// TIA Portal V17 export
// export: Created 2022-07-20T06:59:49.2004828Z, ExportSetting WithDefaults, DisplayName Totally Integrated Automation Portal, DisplayVersion V17, DisplayName TIA Portal Openness, DisplayVersion V17, DisplayName TIA Portal Version Control Interface, DisplayVersion V17, DisplayName SINAMICS Startdrive Advanced, DisplayVersion V17, DisplayName SINAMICS Startdrive G130, G150, S120, S150, SINAMICS MV, S210, DisplayVersion V17, DisplayName SINAMICS Startdrive G110M, G120, G120C, G120D, G120P, G115D, DisplayVersion V17, DisplayName STEP 7 Professional, DisplayVersion V17, DisplayName STEP 7 Safety, DisplayVersion V17, DisplayName WinCC Advanced, DisplayVersion V17
FUNCTION_BLOCK "FB10300_TM_Pulse"   // FB10300, LAD
TITLE = FB10030_TM_Pulse
{ S7_Optimized_Access := 'TRUE' }
AUTHOR : Anirouddh
FAMILY : 1030_SIEMENS
VERSION : 1.0
// Release note : 
// 1.0 - Feature developped
// 
// Todo: 
// - If necessary, complete thre static TM_Pulse structure with the QLMN_HLM & QLMN_LLM to verify that the set value is bounded within the limits
// stored: AutoNumber false, IsIECCheckEnabled false, IsRetainMemResEnabled false, MemoryReserve 100, SetENOAutomatically false, UDAEnableTagReadback false
   VAR_INPUT
      Channel0_SW_Enable : Bool;
      Channel0_Reset_Error : Bool;
      Channel0_Frequency : Real;
      Channel0_Dir : Bool;
      Channel1_SW_Enable : Bool;
      Channel1_Reset_Error : Bool;
      Channel1_Frequency : Real;
      Channel1_Dir : Bool;
      HW_TM_Puls : HW_SUBMODULE;
   END_VAR
   VAR_OUTPUT
      Channel0_Ready : Bool;
      Channel0_SW_Enabled : Bool;
      Channel0_Enable : Bool;
      Channel0_Error : Bool;
      Channel0_DQA : Bool;
      Channel0_Output_Dir : Bool;
      Channel1_Ready : Bool;
      Channel1_SW_Enabled : Bool;
      Channel1_Enable : Bool;
      Channel1_Error : Bool;
      Channel1_DQA : Bool;
      Channel1_Output_Dir : Bool;
   END_VAR
   VAR
      Input_Channel : Array[0..1] of Struct
         ERR_STS1 : Struct
            ERR_PWR : Bool;
            ERR_24V : Bool;
            ERR_LD : Bool;
            ERR_PULSE : Bool;
            ERR_DQA : Bool;
            ERR_DQB : Bool;
            ERR_OUT_VALUE : Bool;
            ERR_SLOT_VAL : Bool;
            Reserved_Bit0 : Bool;
            Reserved_Bit1 : Bool;
            STS_LD_SLOT : Bool;
            Reserved_Bit3 : Bool;
            STS_READY : Bool;
            STS_SW_ENABLE : Bool;
            Reserved_Bit6 : Bool;
            Reserved_Bit7 : Bool;
         END_STRUCT;
         STS2_CNT : Struct
            STS_ENABLE : Bool;
            STS_DQA : Bool;
            STS_DQB : Bool;
            STS_DI : Bool;
            STS_DITHER : Bool;
            Reserved_Bit5 : Bool;
            Reserved_Bit6 : Bool;
            Reserved_Bit7 : Bool;
            SEQ_CNT : Byte;
         END_STRUCT;
         Measured_Current : Word;
         Reserve : Word;
      END_STRUCT;
      Output_Channel : Array[0..1] of Struct
         Output_Value : DWord;
         Slot : DWord;
         Mode_Cmd : Struct
            LD_SLOT_0 : Bool;
            LD_SLOT_1 : Bool;
            LD_SLOT_2 : Bool;
            LD_SLOT_3 : Bool;
            MODE_SLOT : Bool;
            Reserved_Bit5 : Bool;
            Reserved_Bit6 : Bool;
            Reserved_Bit7 : Bool;
            SW_ENABLE : Bool;
            TM_CTRL_DQ : Bool;
            Reserved_Bit2 : Bool;
            SET_DQA : Bool;
            SET_DQB : Bool;
            DITHER : Bool;
            Reserved_Bit8 : Bool;
            Reserved_Bit9 : Bool;
         END_STRUCT;
         Reset : Struct
            RES_ERROR : Bool;
            Reserved_bit1 : Bool;
            Reserved_Bit2 : Bool;
            Reserved_Bit3 : Bool;
            Reserved_Bit4 : Bool;
            Reserved_Bit5 : Bool;
            Reserved_Bit6 : Bool;
            Reserved_Bit7 : Bool;
            Reserved_Bit8 : Bool;
            Reserved_Bit9 : Bool;
            Reserved_Bit10 : Bool;
            Reserved_Bit11 : Bool;
            Reserved_Bit12 : Bool;
            Reserved_Bit13 : Bool;
            Reserved_Bit14 : Bool;
            Reserved_Bit15 : Bool;
         END_STRUCT;
      END_STRUCT;
      RET_VAL_DPRD_DAT : Int;
      RET_VAL_DPWD_DAT : Int;
   END_VAR
BEGIN

REGION Network 1: Read data from TM_Pulse
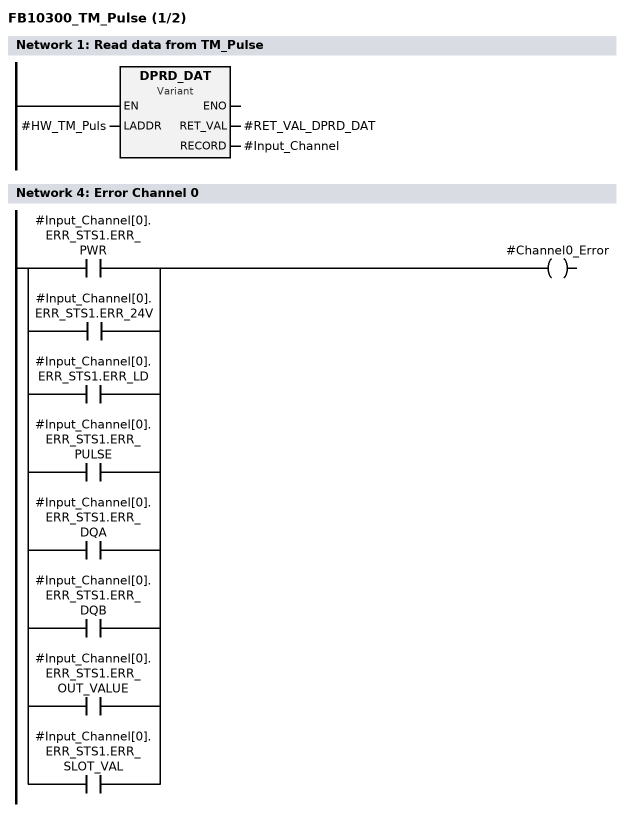
   RUNG wire#powerrail
      { S7_Templates := "[ptr_type := Variant, laddr_type := HW_IO]" } DPRD_DAT(LADDR := #HW_TM_Puls, RET_VAL => #RET_VAL_DPRD_DAT, RECORD => #Input_Channel)
   END_RUNG
   // the same network as SCL:
   #RET_VAL_DPRD_DAT := DPRD_DAT(LADDR := #HW_TM_Puls, RECORD => #Input_Channel);
END_REGION

REGION Network 2 (SCL): Command Channel 0
   #Output_Channel[0].Mode_Cmd.SW_ENABLE := #Channel0_SW_Enable; //Command SW_ENABLE Channel 0
   #Output_Channel[0].Reset.RES_ERROR := #Channel0_Reset_Error; // Command RES_ERROR Channel 0
   #Output_Channel[0].Mode_Cmd.TM_CTRL_DQ := TRUE; //Command TM_CTRL_DQ Channel 0 (The module creates the pulse sequence automatically)
   #Channel0_Output_Dir := #Channel0_Dir; //Command direction Channel 0
   #Output_Channel[0].Output_Value := REAL_TO_DWORD(#Channel0_Frequency); //Command frequence Channel 0

   #Channel0_Ready := #Input_Channel[0].ERR_STS1.STS_READY; //Ready Channel 0
   #Channel0_SW_Enabled := #Input_Channel[0].ERR_STS1.STS_SW_ENABLE; //SW_Enable Channel 0
   #Channel0_Enable := #Input_Channel[0].STS2_CNT.STS_ENABLE; //Enable Channel 0
   #Channel0_DQA := #Input_Channel[0].STS2_CNT.STS_DQA; //DQA Channel 0
END_REGION

REGION Network 3 (SCL): Command Channel 1
   #Output_Channel[1].Mode_Cmd.SW_ENABLE := #Channel1_SW_Enable; //Command SW_ENABLE Channel 1
   #Output_Channel[1].Reset.RES_ERROR := #Channel1_Reset_Error; //Command RES_ERROR Channel 1
   #Output_Channel[1].Mode_Cmd.TM_CTRL_DQ := TRUE; //Command TM_CTRL_DQ Channel 1 (The module creates the pulse sequence automatically)
   #Channel1_Output_Dir := #Channel1_Dir; //Command direction Channel 1
   #Output_Channel[1].Output_Value := REAL_TO_DWORD(#Channel1_Frequency); //Command frequence Channel 1

   #Channel1_Ready := #Input_Channel[1].ERR_STS1.STS_READY; //Ready Channel 1
   #Channel1_SW_Enabled := #Input_Channel[1].ERR_STS1.STS_SW_ENABLE; //SW_Enable Channel 1
   #Channel1_Enable := #Input_Channel[1].STS2_CNT.STS_ENABLE; //Enable Channel 1
   #Channel1_DQA := #Input_Channel[1].STS2_CNT.STS_DQA; //DQA Channel 1
END_REGION

REGION Network 4: Error Channel 0
   RUNG wire#powerrail
      Contact( #Input_Channel[0].ERR_STS1.ERR_PWR )
      wire#w1
      Coil( #Channel0_Error )
   END_RUNG
   RUNG wire#powerrail
      Contact( #Input_Channel[0].ERR_STS1.ERR_24V )
   END_RUNG wire#w1
   RUNG wire#powerrail
      Contact( #Input_Channel[0].ERR_STS1.ERR_LD )
   END_RUNG wire#w1
   RUNG wire#powerrail
      Contact( #Input_Channel[0].ERR_STS1.ERR_PULSE )
   END_RUNG wire#w1
   RUNG wire#powerrail
      Contact( #Input_Channel[0].ERR_STS1.ERR_DQA )
   END_RUNG wire#w1
   RUNG wire#powerrail
      Contact( #Input_Channel[0].ERR_STS1.ERR_DQB )
   END_RUNG wire#w1
   RUNG wire#powerrail
      Contact( #Input_Channel[0].ERR_STS1.ERR_OUT_VALUE )
   END_RUNG wire#w1
   RUNG wire#powerrail
      Contact( #Input_Channel[0].ERR_STS1.ERR_SLOT_VAL )
   END_RUNG wire#w1
   // the same network as SCL:
   #Channel0_Error := #Input_Channel[0].ERR_STS1.ERR_PWR OR #Input_Channel[0].ERR_STS1.ERR_24V OR #Input_Channel[0].ERR_STS1.ERR_LD OR #Input_Channel[0].ERR_STS1.ERR_PULSE OR #Input_Channel[0].ERR_STS1.ERR_DQA OR #Input_Channel[0].ERR_STS1.ERR_DQB OR #Input_Channel[0].ERR_STS1.ERR_OUT_VALUE OR #Input_Channel[0].ERR_STS1.ERR_SLOT_VAL;
END_REGION

REGION Network 5: Error Channel 1
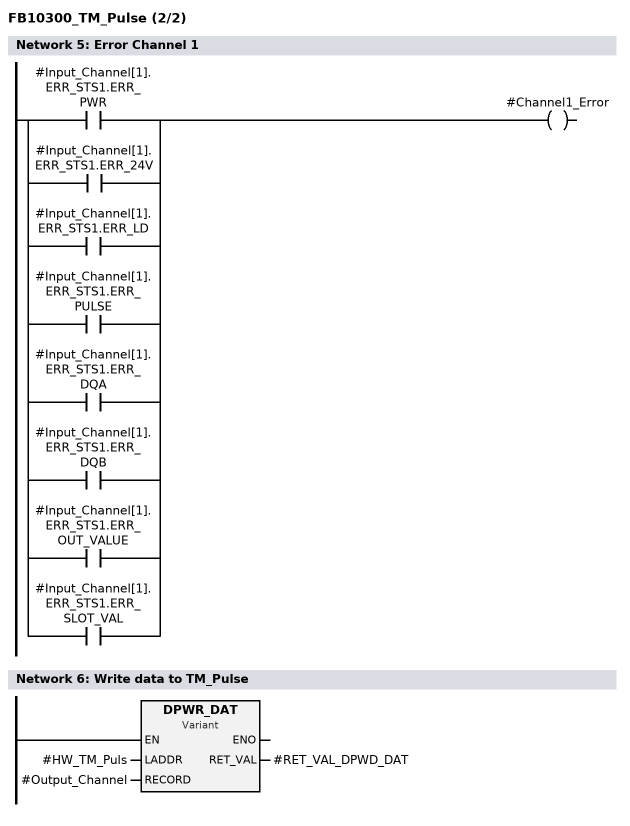
   RUNG wire#powerrail
      Contact( #Input_Channel[1].ERR_STS1.ERR_PWR )
      wire#w1
      Coil( #Channel1_Error )
   END_RUNG
   RUNG wire#powerrail
      Contact( #Input_Channel[1].ERR_STS1.ERR_24V )
   END_RUNG wire#w1
   RUNG wire#powerrail
      Contact( #Input_Channel[1].ERR_STS1.ERR_LD )
   END_RUNG wire#w1
   RUNG wire#powerrail
      Contact( #Input_Channel[1].ERR_STS1.ERR_PULSE )
   END_RUNG wire#w1
   RUNG wire#powerrail
      Contact( #Input_Channel[1].ERR_STS1.ERR_DQA )
   END_RUNG wire#w1
   RUNG wire#powerrail
      Contact( #Input_Channel[1].ERR_STS1.ERR_DQB )
   END_RUNG wire#w1
   RUNG wire#powerrail
      Contact( #Input_Channel[1].ERR_STS1.ERR_OUT_VALUE )
   END_RUNG wire#w1
   RUNG wire#powerrail
      Contact( #Input_Channel[1].ERR_STS1.ERR_SLOT_VAL )
   END_RUNG wire#w1
   // the same network as SCL:
   #Channel1_Error := #Input_Channel[1].ERR_STS1.ERR_PWR OR #Input_Channel[1].ERR_STS1.ERR_24V OR #Input_Channel[1].ERR_STS1.ERR_LD OR #Input_Channel[1].ERR_STS1.ERR_PULSE OR #Input_Channel[1].ERR_STS1.ERR_DQA OR #Input_Channel[1].ERR_STS1.ERR_DQB OR #Input_Channel[1].ERR_STS1.ERR_OUT_VALUE OR #Input_Channel[1].ERR_STS1.ERR_SLOT_VAL;
END_REGION

REGION Network 6: Write data to TM_Pulse
   RUNG wire#powerrail
      { S7_Templates := "[ptr_type := Variant, laddr_type := HW_IO]" } DPWR_DAT(LADDR := #HW_TM_Puls, RECORD := #Output_Channel, RET_VAL => #RET_VAL_DPWD_DAT)
   END_RUNG
   // the same network as SCL:
   #RET_VAL_DPWD_DAT := DPWR_DAT(LADDR := #HW_TM_Puls, RECORD := #Output_Channel);
END_REGION
END_FUNCTION_BLOCK
